Staubli VAL3: return_config.pgx

program return_config(num x_nNum_choose, num& x_nNum_lRow, num& x_nNum_lCol)
begin

   switch x_nNum_choose
    case 1
      //f1
      x_nNum_lCol = 5
      x_nNum_lRow = 5
    break
    case 2
      //f2
      x_nNum_lCol = 11
      x_nNum_lRow = 2
    break
    case 3
      //f3
      //x_nNum_lCol = 2
      //x_nNum_lRow = 5

      x_nNum_lCol = 5
      x_nNum_lRow = 2
    break
    case 4
      //bottom
      x_nNum_lCol = 2
      x_nNum_lRow = 5
    break

  endSwitch

end
